Staubli VAL3: CUTOUT.pgx

public program CutOut(trsf x_trCenter, trsf& x_trLine[], trsf& x_trDest[], trsf& x_trCut, num x_nType, num x_nPercent, bool& x_bRes)
  local trsf l_trTrsf[2]
begin
  //切入引线
    if x_nType==0
    x_bRes=true
    return
    endIf
  call CutIn(x_trCenter,x_trLine,l_trTrsf,x_trCut,x_nType,x_nPercent,x_bRes)
  if !x_bRes
    return
  endIf

  x_trLine[1]=x_trLine[0]
  x_trLine[0]=x_trCenter


  call LineSymArray(l_trTrsf,x_trLine,x_trDest,x_bRes)


end
